FUNCTION_BLOCK AtvResetError_HMI (* Service Interface Function Block Type *)
  (* Standard: 61499-2 *)
  (* Version 0.0, 8/19/2024, SESA713705, Schneider Electric, template *)
  PACKAGE SE.Nereda;
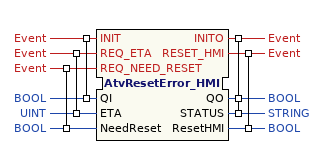
  EVENT_INPUT
    INIT WITH QI;
    REQ_ETA WITH ETA;
    REQ_NEED_RESET WITH NeedReset;
  END_EVENT
  EVENT_OUTPUT
    INITO WITH QO, STATUS;
    RESET_HMI WITH ResetHMI;
  END_EVENT
  VAR_INPUT
    QI : BOOL;
    ETA : UINT;
    NeedReset : BOOL;
  END_VAR
  VAR_OUTPUT
    QO : BOOL; (* Event Output Qualifier *)
    STATUS : STRING; (* Service Status *)
    ResetHMI : BOOL;
  END_VAR
  SERVICE /
    SEQUENCE 
    END_SEQUENCE
  END_SERVICE
END_FUNCTION_BLOCK
